INTERFACE PUBLIC ILog

METHOD SetLogger : BOOL
VAR_INPUT
    ref2Core : ILogCore;
END_VAR
END_METHOD

END_INTERFACE

(* stored: Version 1.1.0.1
   Itf ILog: Id {210033b2-8ae4-4f23-84c0-7b73662b5f23}
   Method SetLogger: Id {feb206be-40e9-4284-a591-4cc26f28a4aa} *)
